(* Logix 5000 project; controller SX_V040001_C001 vendor 1 type 14 code 77 rev 16.23; software revision 16.04; part 8 of 35 *)
(* tags used below, declared in another part *)
   ALL_KINDS : INT[90];
   DRIVE : INT[32];
   DRIVE_INTERVAL : INT[8];
   EMPTYING : INT[18];
   G_DInput : DINT[3];
   loading : INT[19];
   METERING : INT[44];
   PARAMETER : INT[501];
   RECIPE_GENERAL : INT[405];
   TEMP : INT[14];
(* MainProgram, continued *)

ROUTINE AnalyseRecipe   (* ladder *)
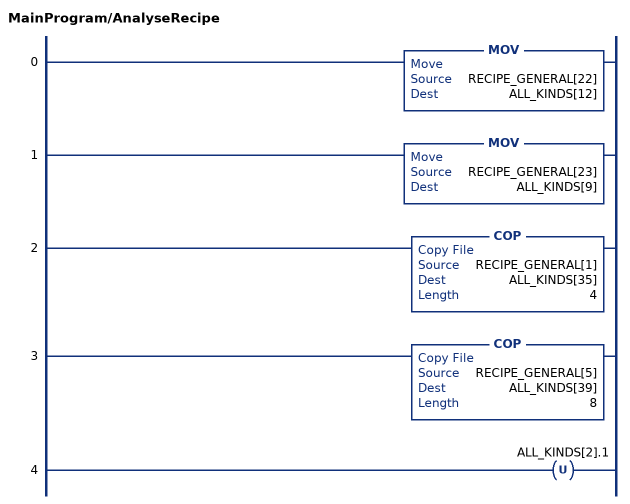
   0: MOV(RECIPE_GENERAL[22],ALL_KINDS[12]);
   1: MOV(RECIPE_GENERAL[23],ALL_KINDS[9]);
   2: COP(RECIPE_GENERAL[1],ALL_KINDS[35],4);
   3: COP(RECIPE_GENERAL[5],ALL_KINDS[39],8);
   4: OTU(ALL_KINDS[2].1);
END_ROUTINE

ROUTINE AnalyseRestart   (* ladder *)
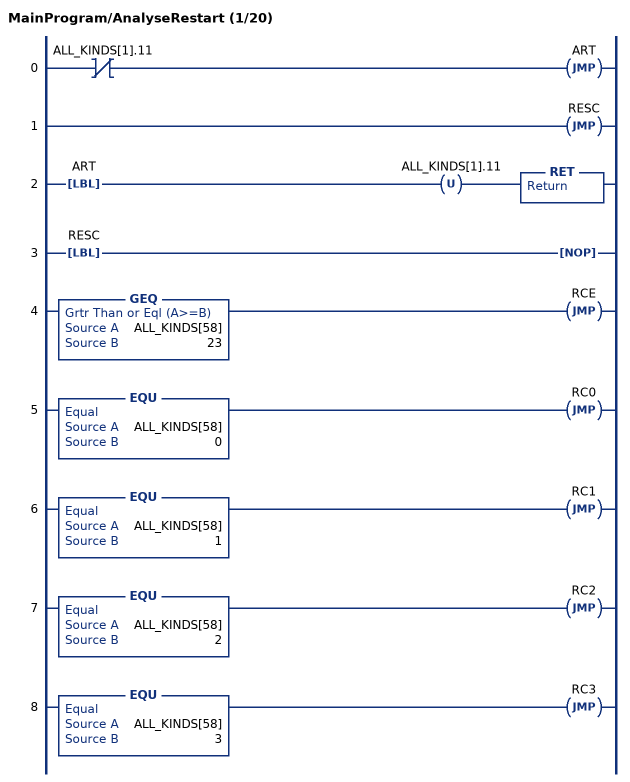
   0: XIO(ALL_KINDS[1].11)JMP(ART);
   1: JMP(RESC);
   2: LBL(ART)OTU(ALL_KINDS[1].11)RET();
   3: LBL(RESC)NOP();
   4: GEQ(ALL_KINDS[58],23)JMP(RCE);
   5: EQU(ALL_KINDS[58],0)JMP(RC0);
   6: EQU(ALL_KINDS[58],1)JMP(RC1);
   7: EQU(ALL_KINDS[58],2)JMP(RC2);
   8: EQU(ALL_KINDS[58],3)JMP(RC3);
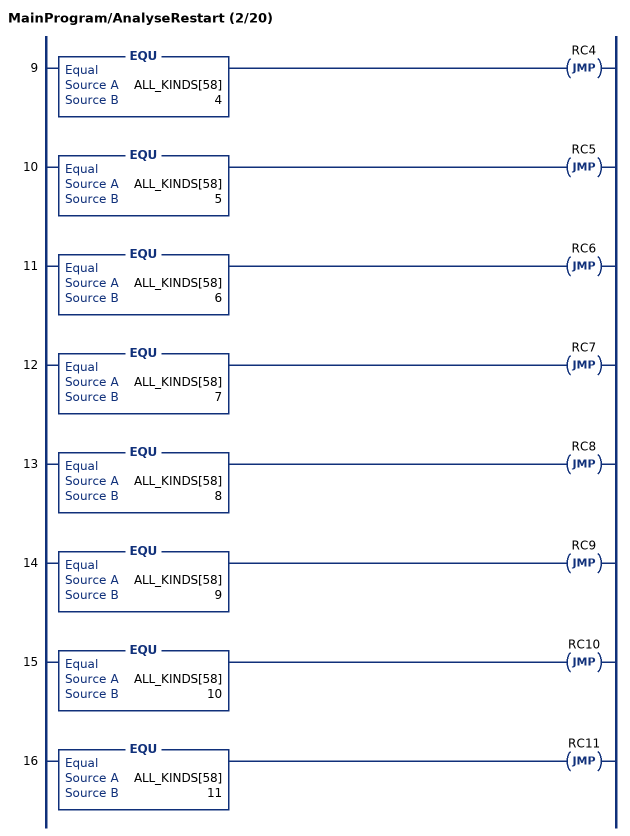
   9: EQU(ALL_KINDS[58],4)JMP(RC4);
   10: EQU(ALL_KINDS[58],5)JMP(RC5);
   11: EQU(ALL_KINDS[58],6)JMP(RC6);
   12: EQU(ALL_KINDS[58],7)JMP(RC7);
   13: EQU(ALL_KINDS[58],8)JMP(RC8);
   14: EQU(ALL_KINDS[58],9)JMP(RC9);
   15: EQU(ALL_KINDS[58],10)JMP(RC10);
   16: EQU(ALL_KINDS[58],11)JMP(RC11);
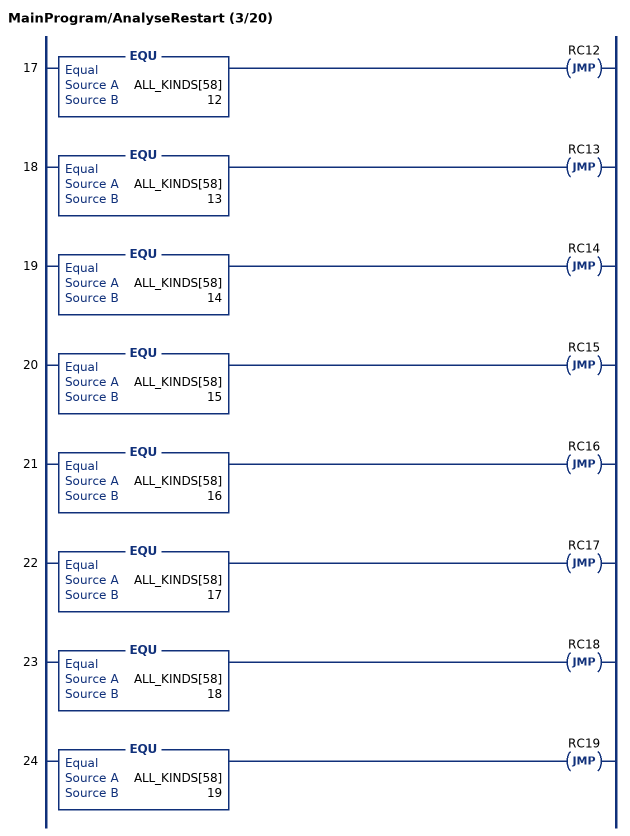
   17: EQU(ALL_KINDS[58],12)JMP(RC12);
   18: EQU(ALL_KINDS[58],13)JMP(RC13);
   19: EQU(ALL_KINDS[58],14)JMP(RC14);
   20: EQU(ALL_KINDS[58],15)JMP(RC15);
   21: EQU(ALL_KINDS[58],16)JMP(RC16);
   22: EQU(ALL_KINDS[58],17)JMP(RC17);
   23: EQU(ALL_KINDS[58],18)JMP(RC18);
   24: EQU(ALL_KINDS[58],19)JMP(RC19);
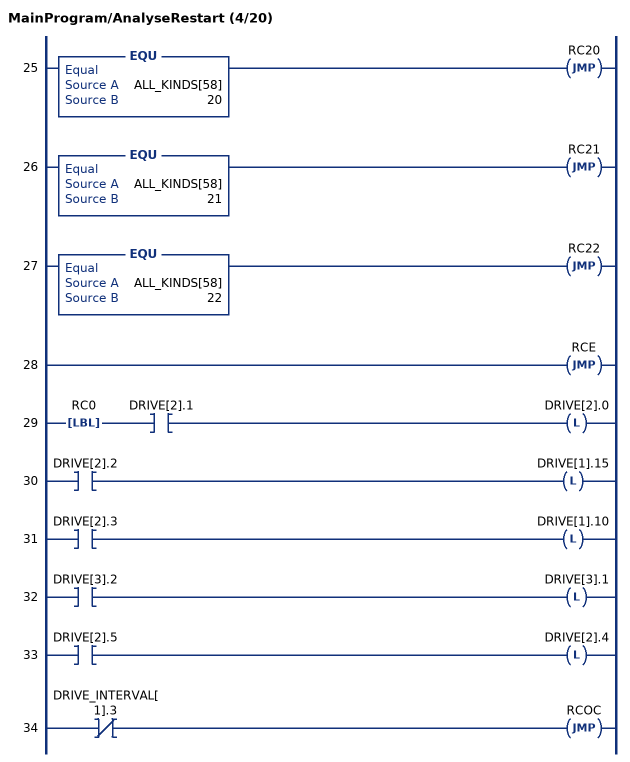
   25: EQU(ALL_KINDS[58],20)JMP(RC20);
   26: EQU(ALL_KINDS[58],21)JMP(RC21);
   27: EQU(ALL_KINDS[58],22)JMP(RC22);
   28: JMP(RCE);
   29: LBL(RC0)XIC(DRIVE[2].1)OTL(DRIVE[2].0);
   30: XIC(DRIVE[2].2)OTL(DRIVE[1].15);
   31: XIC(DRIVE[2].3)OTL(DRIVE[1].10);
   32: XIC(DRIVE[3].2)OTL(DRIVE[3].1);
   33: XIC(DRIVE[2].5)OTL(DRIVE[2].4);
   34: XIO(DRIVE_INTERVAL[1].3)JMP(RCOC);
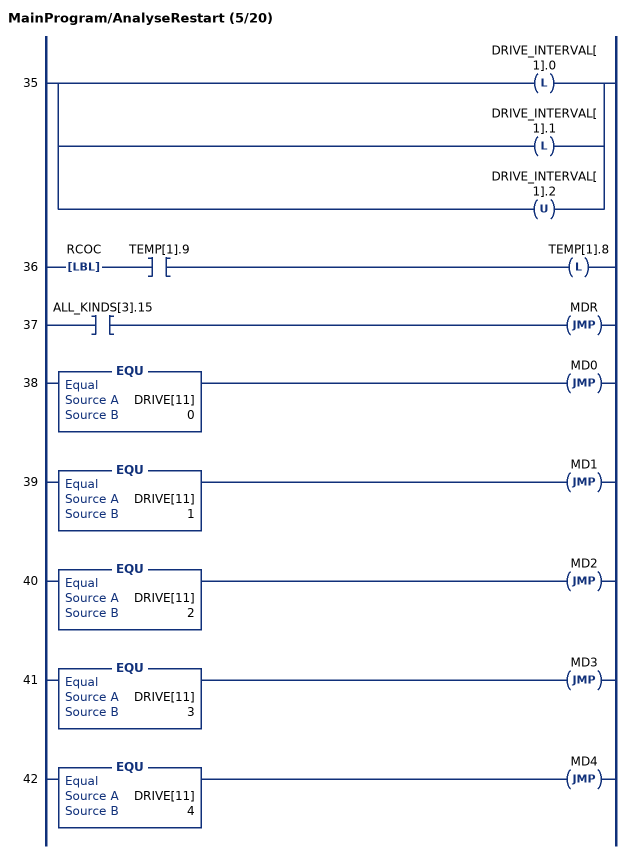
   35: [OTL(DRIVE_INTERVAL[1].0) ,OTL(DRIVE_INTERVAL[1].1) ,OTU(DRIVE_INTERVAL[1].2) ];
   36: LBL(RCOC)XIC(TEMP[1].9)OTL(TEMP[1].8);
   37: XIC(ALL_KINDS[3].15)JMP(MDR);
   38: EQU(DRIVE[11],0)JMP(MD0);
   39: EQU(DRIVE[11],1)JMP(MD1);
   40: EQU(DRIVE[11],2)JMP(MD2);
   41: EQU(DRIVE[11],3)JMP(MD3);
   42: EQU(DRIVE[11],4)JMP(MD4);
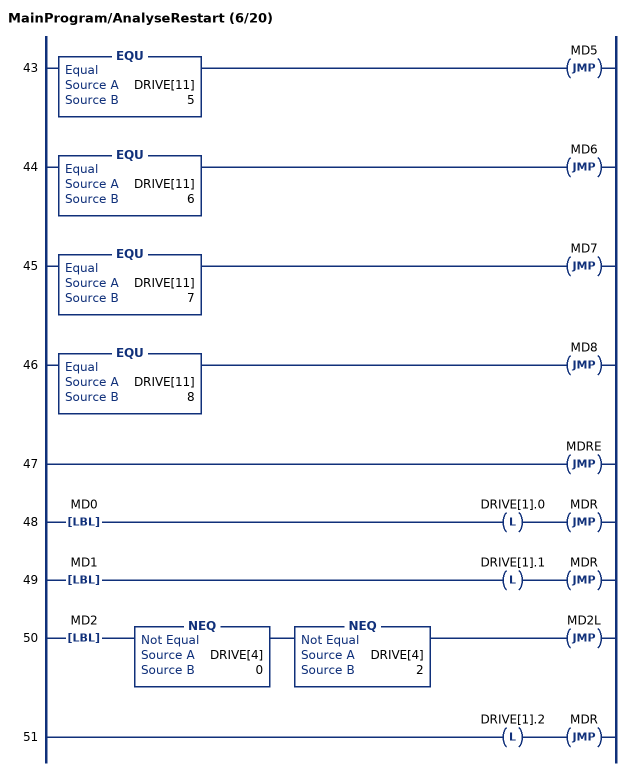
   43: EQU(DRIVE[11],5)JMP(MD5);
   44: EQU(DRIVE[11],6)JMP(MD6);
   45: EQU(DRIVE[11],7)JMP(MD7);
   46: EQU(DRIVE[11],8)JMP(MD8);
   47: JMP(MDRE);
   48: LBL(MD0)OTL(DRIVE[1].0)JMP(MDR);
   49: LBL(MD1)OTL(DRIVE[1].1)JMP(MDR);
   50: LBL(MD2)NEQ(DRIVE[4],0)NEQ(DRIVE[4],2)JMP(MD2L);
   51: OTL(DRIVE[1].2)JMP(MDR);
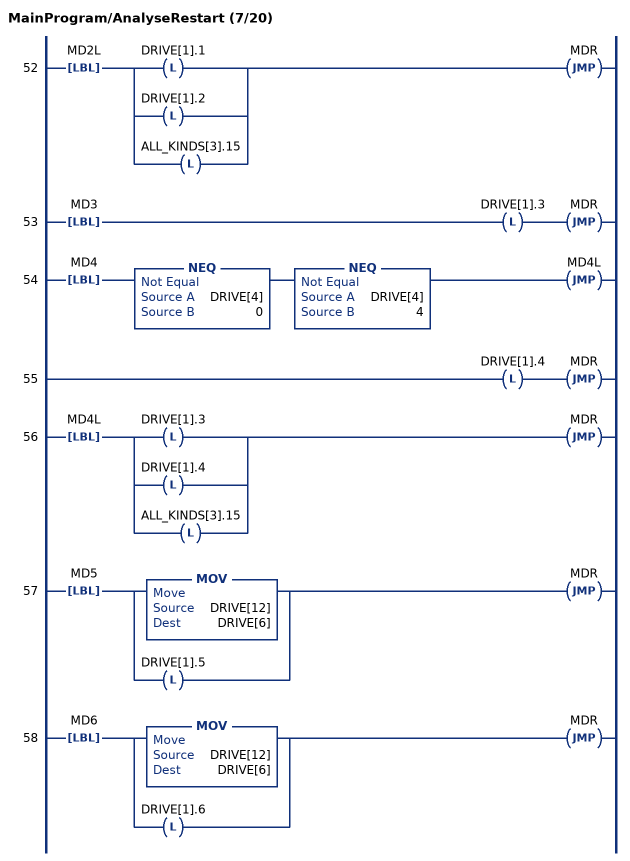
   52: LBL(MD2L)[OTL(DRIVE[1].1) ,OTL(DRIVE[1].2) ,OTL(ALL_KINDS[3].15) ]JMP(MDR);
   53: LBL(MD3)OTL(DRIVE[1].3)JMP(MDR);
   54: LBL(MD4)NEQ(DRIVE[4],0)NEQ(DRIVE[4],4)JMP(MD4L);
   55: OTL(DRIVE[1].4)JMP(MDR);
   56: LBL(MD4L)[OTL(DRIVE[1].3) ,OTL(DRIVE[1].4) ,OTL(ALL_KINDS[3].15) ]JMP(MDR);
   57: LBL(MD5)[MOV(DRIVE[12],DRIVE[6]) ,OTL(DRIVE[1].5) ]JMP(MDR);
   58: LBL(MD6)[MOV(DRIVE[12],DRIVE[6]) ,OTL(DRIVE[1].6) ]JMP(MDR);
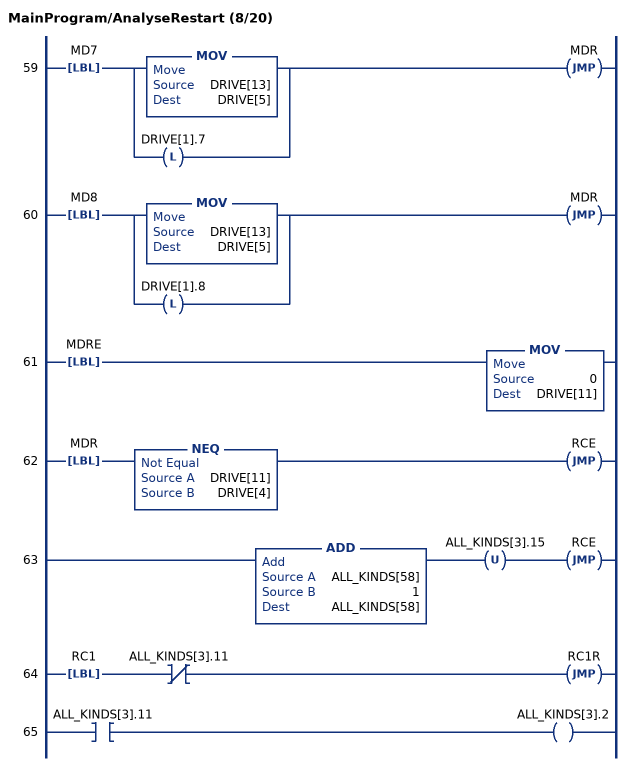
   59: LBL(MD7)[MOV(DRIVE[13],DRIVE[5]) ,OTL(DRIVE[1].7) ]JMP(MDR);
   60: LBL(MD8)[MOV(DRIVE[13],DRIVE[5]) ,OTL(DRIVE[1].8) ]JMP(MDR);
   61: LBL(MDRE)MOV(0,DRIVE[11]);
   62: LBL(MDR)NEQ(DRIVE[11],DRIVE[4])JMP(RCE);
   63: ADD(ALL_KINDS[58],1,ALL_KINDS[58])OTU(ALL_KINDS[3].15)JMP(RCE);
   64: LBL(RC1)XIO(ALL_KINDS[3].11)JMP(RC1R);
   65: XIC(ALL_KINDS[3].11)OTE(ALL_KINDS[3].2);
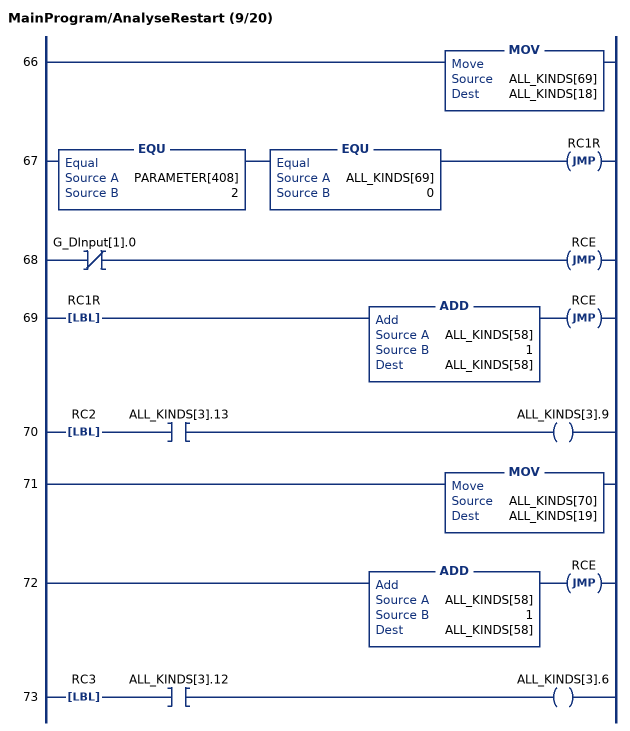
   66: MOV(ALL_KINDS[69],ALL_KINDS[18]);
   67: EQU(PARAMETER[408],2)EQU(ALL_KINDS[69],0)JMP(RC1R);
   68: XIO(G_DInput[1].0)JMP(RCE);
   69: LBL(RC1R)ADD(ALL_KINDS[58],1,ALL_KINDS[58])JMP(RCE);
   70: LBL(RC2)XIC(ALL_KINDS[3].13)OTE(ALL_KINDS[3].9);
   71: MOV(ALL_KINDS[70],ALL_KINDS[19]);
   72: ADD(ALL_KINDS[58],1,ALL_KINDS[58])JMP(RCE);
   73: LBL(RC3)XIC(ALL_KINDS[3].12)OTE(ALL_KINDS[3].6);
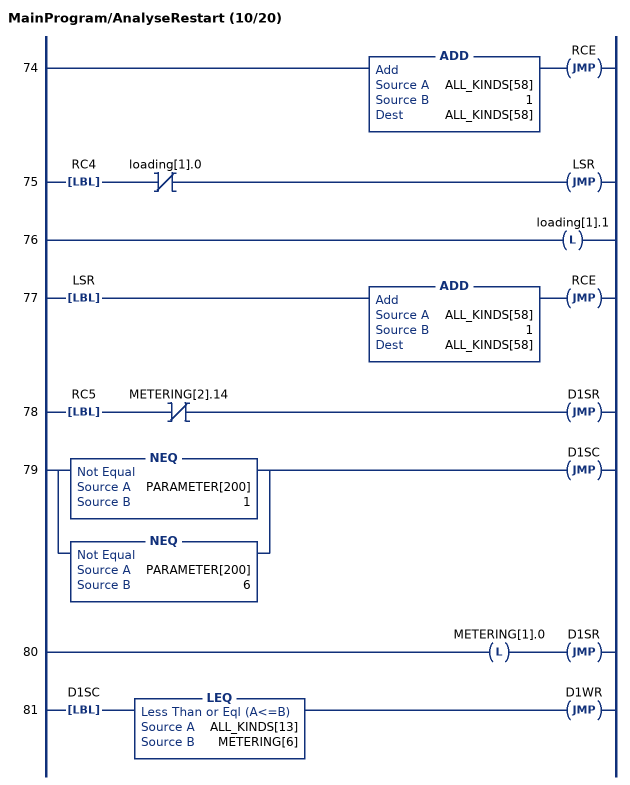
   74: ADD(ALL_KINDS[58],1,ALL_KINDS[58])JMP(RCE);
   75: LBL(RC4)XIO(loading[1].0)JMP(LSR);
   76: OTL(loading[1].1);
   77: LBL(LSR)ADD(ALL_KINDS[58],1,ALL_KINDS[58])JMP(RCE);
   78: LBL(RC5)XIO(METERING[2].14)JMP(D1SR);
   79: [NEQ(PARAMETER[200],1) ,NEQ(PARAMETER[200],6) ]JMP(D1SC);
   80: OTL(METERING[1].0)JMP(D1SR);
   81: LBL(D1SC)LEQ(ALL_KINDS[13],METERING[6])JMP(D1WR);
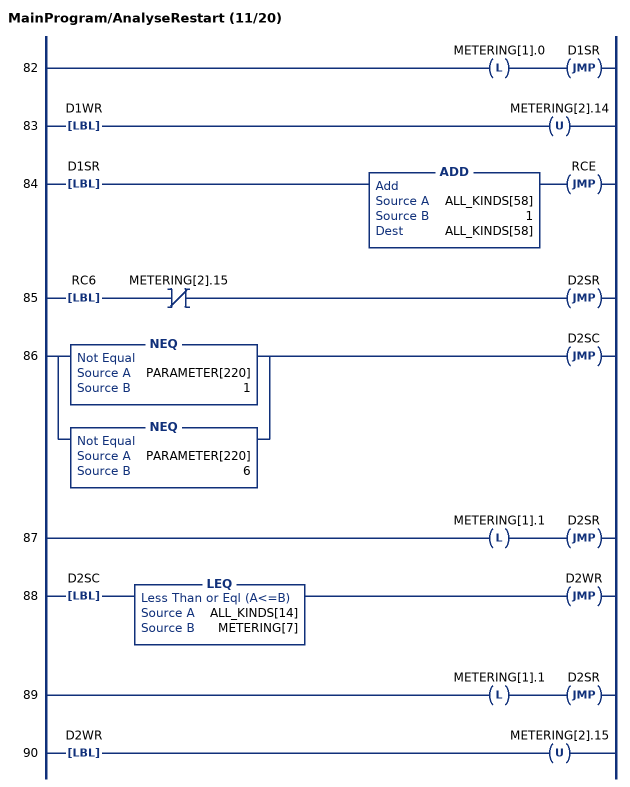
   82: OTL(METERING[1].0)JMP(D1SR);
   83: LBL(D1WR)OTU(METERING[2].14);
   84: LBL(D1SR)ADD(ALL_KINDS[58],1,ALL_KINDS[58])JMP(RCE);
   85: LBL(RC6)XIO(METERING[2].15)JMP(D2SR);
   86: [NEQ(PARAMETER[220],1) ,NEQ(PARAMETER[220],6) ]JMP(D2SC);
   87: OTL(METERING[1].1)JMP(D2SR);
   88: LBL(D2SC)LEQ(ALL_KINDS[14],METERING[7])JMP(D2WR);
   89: OTL(METERING[1].1)JMP(D2SR);
   90: LBL(D2WR)OTU(METERING[2].15);
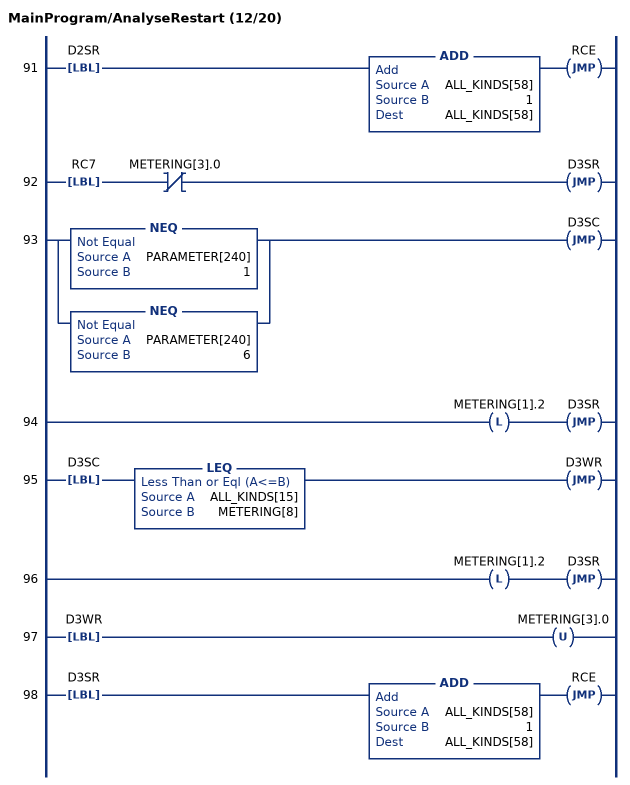
   91: LBL(D2SR)ADD(ALL_KINDS[58],1,ALL_KINDS[58])JMP(RCE);
   92: LBL(RC7)XIO(METERING[3].0)JMP(D3SR);
   93: [NEQ(PARAMETER[240],1) ,NEQ(PARAMETER[240],6) ]JMP(D3SC);
   94: OTL(METERING[1].2)JMP(D3SR);
   95: LBL(D3SC)LEQ(ALL_KINDS[15],METERING[8])JMP(D3WR);
   96: OTL(METERING[1].2)JMP(D3SR);
   97: LBL(D3WR)OTU(METERING[3].0);
   98: LBL(D3SR)ADD(ALL_KINDS[58],1,ALL_KINDS[58])JMP(RCE);
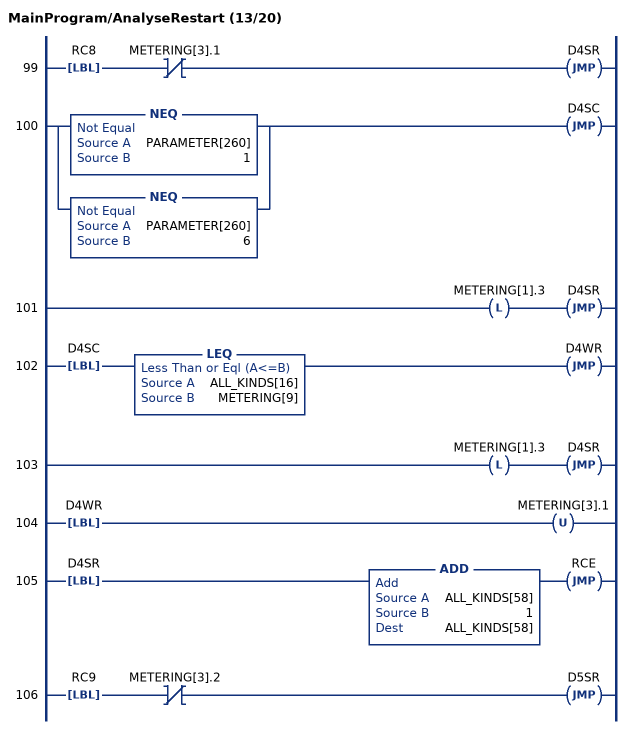
   99: LBL(RC8)XIO(METERING[3].1)JMP(D4SR);
   100: [NEQ(PARAMETER[260],1) ,NEQ(PARAMETER[260],6) ]JMP(D4SC);
   101: OTL(METERING[1].3)JMP(D4SR);
   102: LBL(D4SC)LEQ(ALL_KINDS[16],METERING[9])JMP(D4WR);
   103: OTL(METERING[1].3)JMP(D4SR);
   104: LBL(D4WR)OTU(METERING[3].1);
   105: LBL(D4SR)ADD(ALL_KINDS[58],1,ALL_KINDS[58])JMP(RCE);
   106: LBL(RC9)XIO(METERING[3].2)JMP(D5SR);
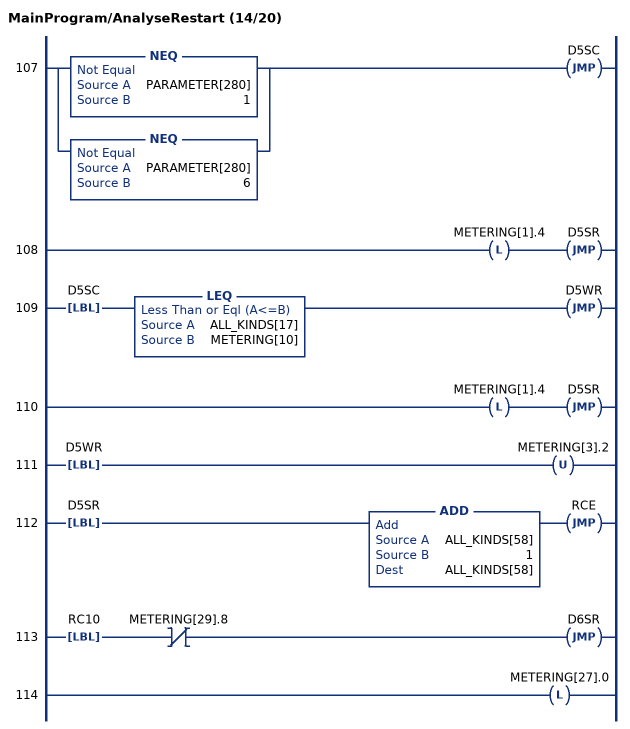
   107: [NEQ(PARAMETER[280],1) ,NEQ(PARAMETER[280],6) ]JMP(D5SC);
   108: OTL(METERING[1].4)JMP(D5SR);
   109: LBL(D5SC)LEQ(ALL_KINDS[17],METERING[10])JMP(D5WR);
   110: OTL(METERING[1].4)JMP(D5SR);
   111: LBL(D5WR)OTU(METERING[3].2);
   112: LBL(D5SR)ADD(ALL_KINDS[58],1,ALL_KINDS[58])JMP(RCE);
   113: LBL(RC10)XIO(METERING[29].8)JMP(D6SR);
   114: OTL(METERING[27].0);
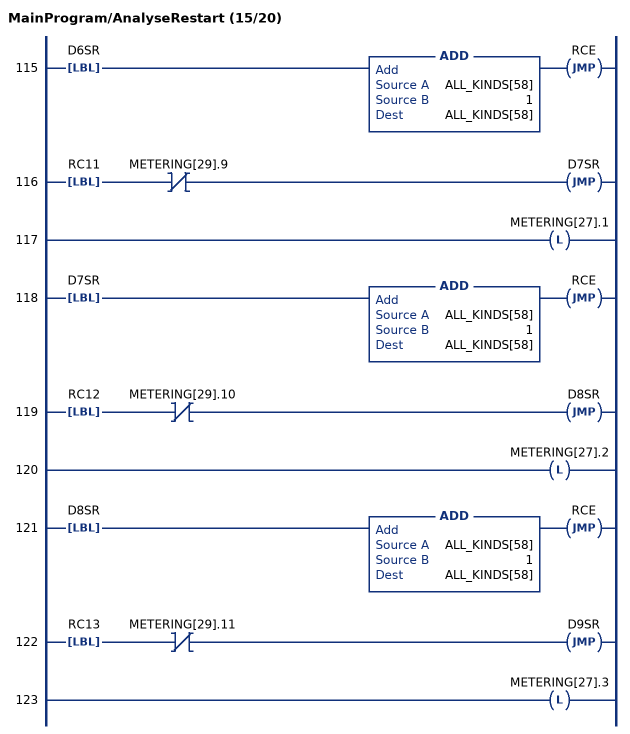
   115: LBL(D6SR)ADD(ALL_KINDS[58],1,ALL_KINDS[58])JMP(RCE);
   116: LBL(RC11)XIO(METERING[29].9)JMP(D7SR);
   117: OTL(METERING[27].1);
   118: LBL(D7SR)ADD(ALL_KINDS[58],1,ALL_KINDS[58])JMP(RCE);
   119: LBL(RC12)XIO(METERING[29].10)JMP(D8SR);
   120: OTL(METERING[27].2);
   121: LBL(D8SR)ADD(ALL_KINDS[58],1,ALL_KINDS[58])JMP(RCE);
   122: LBL(RC13)XIO(METERING[29].11)JMP(D9SR);
   123: OTL(METERING[27].3);
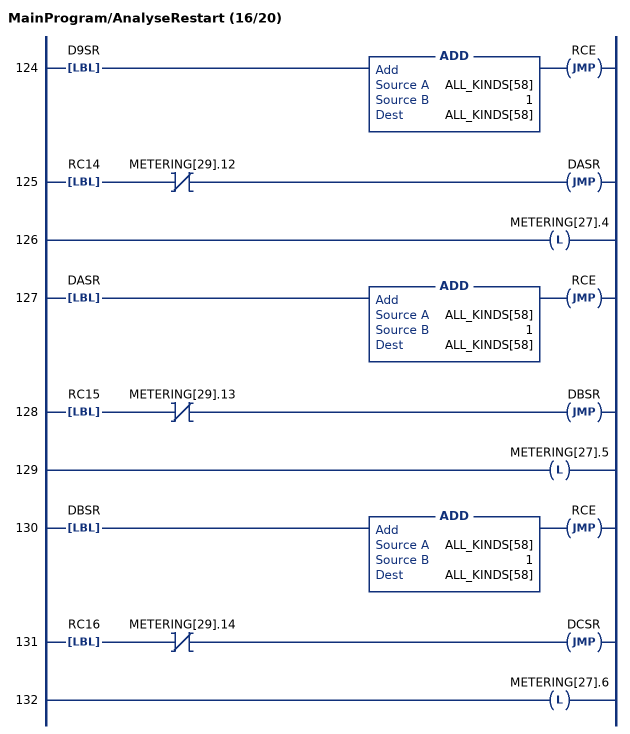
   124: LBL(D9SR)ADD(ALL_KINDS[58],1,ALL_KINDS[58])JMP(RCE);
   125: LBL(RC14)XIO(METERING[29].12)JMP(DASR);
   126: OTL(METERING[27].4);
   127: LBL(DASR)ADD(ALL_KINDS[58],1,ALL_KINDS[58])JMP(RCE);
   128: LBL(RC15)XIO(METERING[29].13)JMP(DBSR);
   129: OTL(METERING[27].5);
   130: LBL(DBSR)ADD(ALL_KINDS[58],1,ALL_KINDS[58])JMP(RCE);
   131: LBL(RC16)XIO(METERING[29].14)JMP(DCSR);
   132: OTL(METERING[27].6);
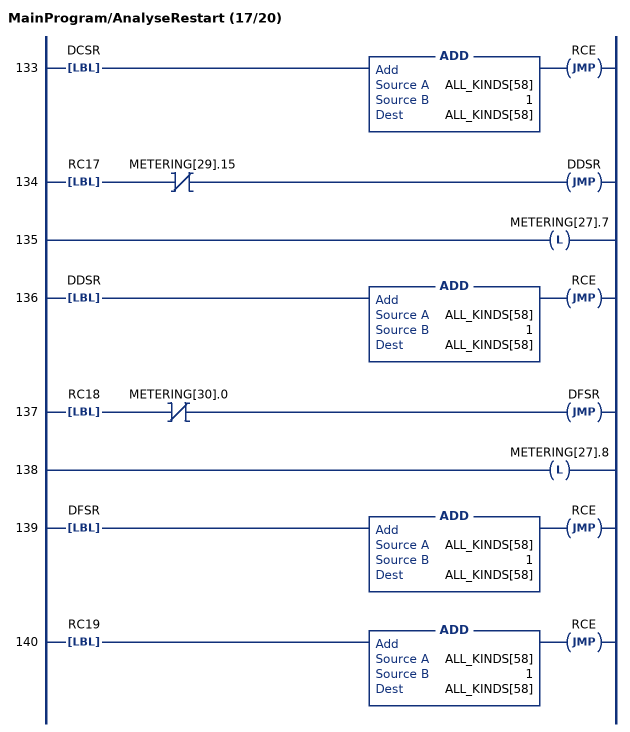
   133: LBL(DCSR)ADD(ALL_KINDS[58],1,ALL_KINDS[58])JMP(RCE);
   134: LBL(RC17)XIO(METERING[29].15)JMP(DDSR);
   135: OTL(METERING[27].7);
   136: LBL(DDSR)ADD(ALL_KINDS[58],1,ALL_KINDS[58])JMP(RCE);
   137: LBL(RC18)XIO(METERING[30].0)JMP(DFSR);
   138: OTL(METERING[27].8);
   139: LBL(DFSR)ADD(ALL_KINDS[58],1,ALL_KINDS[58])JMP(RCE);
   140: LBL(RC19)ADD(ALL_KINDS[58],1,ALL_KINDS[58])JMP(RCE);
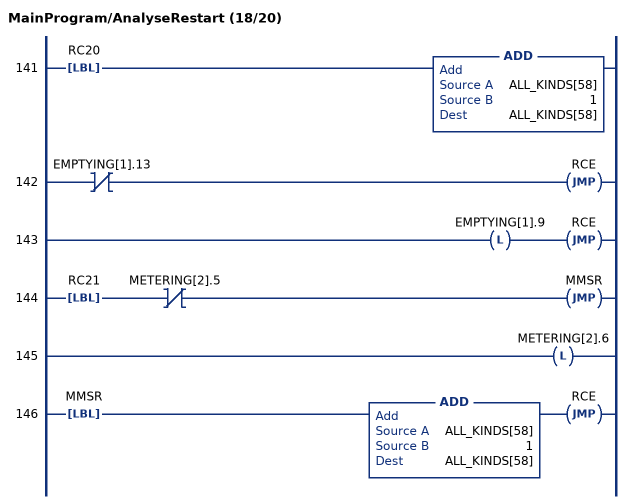
   141: LBL(RC20)ADD(ALL_KINDS[58],1,ALL_KINDS[58]);
   142: XIO(EMPTYING[1].13)JMP(RCE);
   143: OTL(EMPTYING[1].9)JMP(RCE);
   144: LBL(RC21)XIO(METERING[2].5)JMP(MMSR);
   145: OTL(METERING[2].6);
   146: LBL(MMSR)ADD(ALL_KINDS[58],1,ALL_KINDS[58])JMP(RCE);
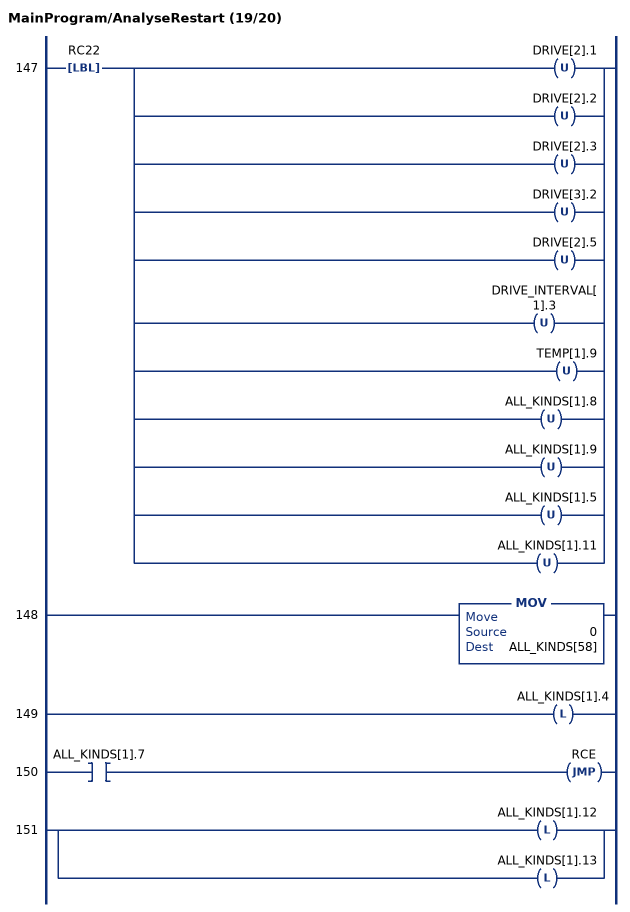
   147: LBL(RC22)[OTU(DRIVE[2].1) ,OTU(DRIVE[2].2) ,OTU(DRIVE[2].3) ,OTU(DRIVE[3].2) ,OTU(DRIVE[2].5) ,OTU(DRIVE_INTERVAL[1].3) ,OTU(TEMP[1].9) ,OTU(ALL_KINDS[1].8) ,OTU(ALL_KINDS[1].9) ,OTU(ALL_KINDS[1].5) ,OTU(ALL_KINDS[1].11) ];
   148: MOV(0,ALL_KINDS[58]);
   149: OTL(ALL_KINDS[1].4);
   150: XIC(ALL_KINDS[1].7)JMP(RCE);
   151: [OTL(ALL_KINDS[1].12) ,OTL(ALL_KINDS[1].13) ];
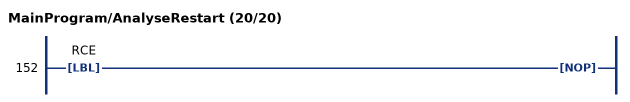
   152: LBL(RCE)NOP();
END_ROUTINE
